Staubli VAL3: recvPacket.pgx

program recvPacket(num& x_nBuff[], num x_nSize)
begin

  resize(nTempBuffer,1,1)
  nTempBuffer=0
  resize(nTempBuffer,1,x_nSize)

  if sioGet(sioTCPclient,nTempBuffer)!=x_nSize
    call setLastError(nErrTCPConnRst)
  endIf

  getData("nTempBuffer",x_nBuff)

end
